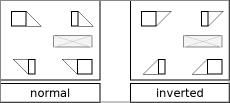
VISUALIZATION _VISU_MarkOrientation  // 230x103
VAR_IN_OUT
  mInst : FB_MarkCamera_WEU;
END_VAR
    RoundedRectangle (0,83 100x20), "normal", colour toggle: NOT mInst.bMarkInverted
        OnMouseClick: execute { mInst.bMarkInverted := FALSE; }
    RoundedRectangle (130,83 100x20), "inverted", colour toggle: mInst.bMarkInverted
        OnMouseClick: execute { mInst.bMarkInverted := TRUE; }
    Rectangle (130,0 100x80), colour toggle: mInst.bMarkInverted
    Image (183,35 39x12), image: VisuSymbols.Symbols.ArrowBoldLeft
    Group (141,11 30x15), invisible if: mInst.bPrintDirReverse
        Polygon (15,0) (15,15) (30,0)
        Rectangle (0,0 15x15)
    Group (201,11 22x15), invisible if: mInst.bPrintDirReverse
        Rectangle (0,0 7x15)
        Polygon (7,0) (7,15) (22,0)
    Rectangle (0,0 100x80), colour toggle: NOT mInst.bMarkInverted
    Image (53,35 39x12), image: VisuSymbols.Symbols.ArrowBoldLeft
    Group (11,11 30x15), invisible if: mInst.bPrintDirReverse
        Polygon (15,0) (15,15) (30,15)
        Rectangle (0,0 15x15)
    Group (71,11 22x15), invisible if: mInst.bPrintDirReverse
        Rectangle (0,0 7x15)
        Polygon (7,0) (7,15) (22,15)
    Group (62,59 30x15), invisible if: NOT mInst.bPrintDirReverse
        Polygon (0,0) (15,15) (15,0)
        Rectangle (15,0 15x15)
    Group (13,59 22x15), invisible if: NOT mInst.bPrintDirReverse
        Rectangle (15,0 7x15)
        Polygon (0,0) (15,15) (15,0)
    Group (192,59 30x15), invisible if: NOT mInst.bPrintDirReverse
        Polygon (0,15) (15,15) (15,0)
        Rectangle (15,0 15x15)
    Group (143,59 22x15), invisible if: NOT mInst.bPrintDirReverse
        Rectangle (15,0 7x15)
        Polygon (0,15) (15,15) (15,0)
END_VISUALIZATION

(* stored: Version 1.1.0.1, ProductVersion 3.1.4024.11
   Visu _VISU_MarkOrientation: Id {558966b3-2504-4d15-814d-9fa207b79ac8} *)
